TYPE Appdata :
STRUCT
		
END_STRUCT
	
END_TYPE

(* stored: Version 1.1.0.1, ProductVersion 3.1.4024.12
   DUT Appdata: Id {874858ec-6b60-44e7-a77b-f6bbbb18ad5b} *)
